// TIA Portal project "SyncProcessi" (V16)

(* hardware
DEVICE "S7-1200 station_1"  S7-1200 Station
   slot 0: "Telaio di montaggio_0"  S7-1200 Rack  Rack  V1.0
   slot 1: "PLC_1"  CPU 1214C DC/DC/DC  6ES7 214-1AG40-0XB0  V4.1
*)

// ===== PLC "PLC_1"  CPU 1214C DC/DC/DC =====

VAR_GLOBAL   // PLC tag table "Tabella delle variabili standard"
   "START_1" AT %I0.0 : Bool;
   "START_2" AT %I0.1 : Bool;
   "STOP_1" AT %I0.2 : Bool;
   "RESTART_2" AT %I0.5 : Bool;
   "OUT_1" AT %Q0.0 : Bool;
   "OUT_2" AT %Q0.1 : Bool;
   "STOP_2" AT %I0.3 : Bool;
   "RESTART_1" AT %I0.4 : Bool;
END_VAR

DATA_BLOCK "VariabiliDiStato_P1"   // DB1
{ S7_Optimized_Access := 'TRUE' }
VERSION : 0.1
   VAR RETAIN
      HOME_1 : Bool := true;
      MOVE : Bool;
      WAIT_1 : Bool;
   END_VAR
BEGIN
END_DATA_BLOCK

DATA_BLOCK "VariabiliDiStato_P2"   // DB2
{ S7_Optimized_Access := 'TRUE' }
VERSION : 0.1
   VAR RETAIN
      HOME_2 : Bool := true;
      ROTATE : Bool;
      WAIT_2 : Bool;
   END_VAR
BEGIN
END_DATA_BLOCK

ORGANIZATION_BLOCK "Main_P1"   // OB1, LAD, ProgramCycle
TITLE = "Main Program Sweep (Cycle)"
{ S7_Optimized_Access := 'TRUE' }
VERSION : 0.1
   VAR_INPUT
      Initial_Call : Bool;   // Initial call of this OB
      Remanence : Bool;   // =True, if remanent data are available
   END_VAR
BEGIN

REGION Network 1
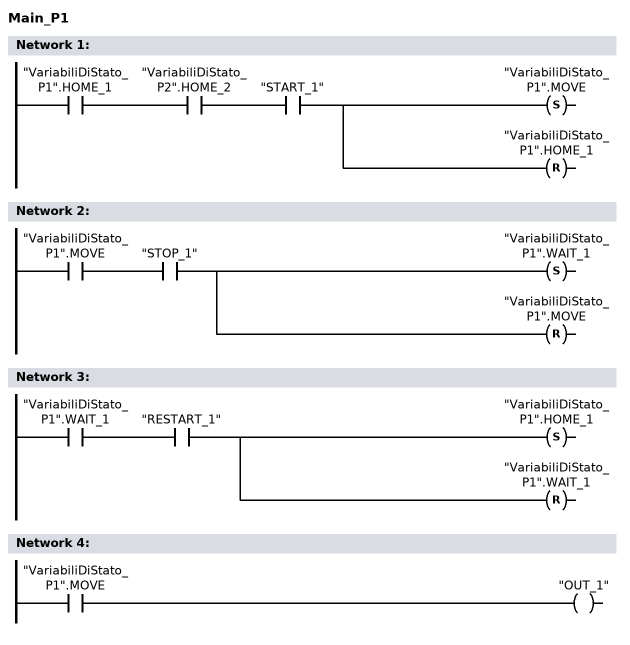
   RUNG wire#powerrail
      Contact( "VariabiliDiStato_P1".HOME_1 )
      Contact( "VariabiliDiStato_P2".HOME_2 )
      Contact( "START_1" )
      wire#w1
      S_Coil( "VariabiliDiStato_P1".MOVE )
   END_RUNG
   RUNG wire#w1
      R_Coil( "VariabiliDiStato_P1".HOME_1 )
   END_RUNG
   // the same network as SCL:
   IF "VariabiliDiStato_P1".HOME_1 AND "VariabiliDiStato_P2".HOME_2 AND "START_1" THEN
       "VariabiliDiStato_P1".MOVE := TRUE;
       "VariabiliDiStato_P1".HOME_1 := FALSE;
   END_IF;
END_REGION

REGION Network 2
   RUNG wire#powerrail
      Contact( "VariabiliDiStato_P1".MOVE )
      Contact( "STOP_1" )
      wire#w1
      S_Coil( "VariabiliDiStato_P1".WAIT_1 )
   END_RUNG
   RUNG wire#w1
      R_Coil( "VariabiliDiStato_P1".MOVE )
   END_RUNG
   // the same network as SCL:
   IF "VariabiliDiStato_P1".MOVE AND "STOP_1" THEN
       "VariabiliDiStato_P1".WAIT_1 := TRUE;
       "VariabiliDiStato_P1".MOVE := FALSE;
   END_IF;
END_REGION

REGION Network 3
   RUNG wire#powerrail
      Contact( "VariabiliDiStato_P1".WAIT_1 )
      Contact( "RESTART_1" )
      wire#w1
      S_Coil( "VariabiliDiStato_P1".HOME_1 )
   END_RUNG
   RUNG wire#w1
      R_Coil( "VariabiliDiStato_P1".WAIT_1 )
   END_RUNG
   // the same network as SCL:
   IF "VariabiliDiStato_P1".WAIT_1 AND "RESTART_1" THEN
       "VariabiliDiStato_P1".HOME_1 := TRUE;
       "VariabiliDiStato_P1".WAIT_1 := FALSE;
   END_IF;
END_REGION

REGION Network 4
   RUNG wire#powerrail
      Contact( "VariabiliDiStato_P1".MOVE )
      Coil( "OUT_1" )
   END_RUNG
   // the same network as SCL:
   "OUT_1" := "VariabiliDiStato_P1".MOVE;
END_REGION
END_ORGANIZATION_BLOCK

ORGANIZATION_BLOCK "Main_P2"   // OB123, LAD, ProgramCycle
TITLE = "Main Program Sweep (Cycle)"
{ S7_Optimized_Access := 'TRUE' }
VERSION : 0.1
   VAR_INPUT
      Initial_Call : Bool;   // Initial call of this OB
      Remanence : Bool;   // =True, if remanent data are available
   END_VAR
BEGIN

REGION Network 1
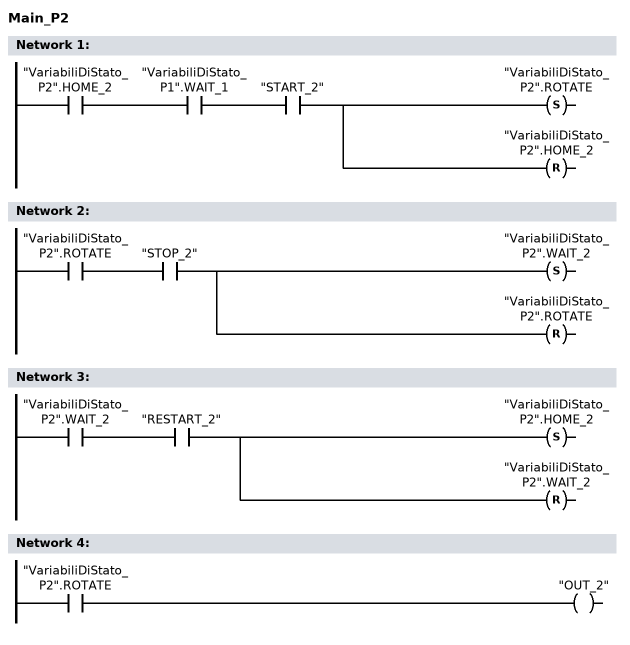
   RUNG wire#powerrail
      Contact( "VariabiliDiStato_P2".HOME_2 )
      Contact( "VariabiliDiStato_P1".WAIT_1 )
      Contact( "START_2" )
      wire#w1
      S_Coil( "VariabiliDiStato_P2".ROTATE )
   END_RUNG
   RUNG wire#w1
      R_Coil( "VariabiliDiStato_P2".HOME_2 )
   END_RUNG
   // the same network as SCL:
   IF "VariabiliDiStato_P2".HOME_2 AND "VariabiliDiStato_P1".WAIT_1 AND "START_2" THEN
       "VariabiliDiStato_P2".ROTATE := TRUE;
       "VariabiliDiStato_P2".HOME_2 := FALSE;
   END_IF;
END_REGION

REGION Network 2
   RUNG wire#powerrail
      Contact( "VariabiliDiStato_P2".ROTATE )
      Contact( "STOP_2" )
      wire#w1
      S_Coil( "VariabiliDiStato_P2".WAIT_2 )
   END_RUNG
   RUNG wire#w1
      R_Coil( "VariabiliDiStato_P2".ROTATE )
   END_RUNG
   // the same network as SCL:
   IF "VariabiliDiStato_P2".ROTATE AND "STOP_2" THEN
       "VariabiliDiStato_P2".WAIT_2 := TRUE;
       "VariabiliDiStato_P2".ROTATE := FALSE;
   END_IF;
END_REGION

REGION Network 3
   RUNG wire#powerrail
      Contact( "VariabiliDiStato_P2".WAIT_2 )
      Contact( "RESTART_2" )
      wire#w1
      S_Coil( "VariabiliDiStato_P2".HOME_2 )
   END_RUNG
   RUNG wire#w1
      R_Coil( "VariabiliDiStato_P2".WAIT_2 )
   END_RUNG
   // the same network as SCL:
   IF "VariabiliDiStato_P2".WAIT_2 AND "RESTART_2" THEN
       "VariabiliDiStato_P2".HOME_2 := TRUE;
       "VariabiliDiStato_P2".WAIT_2 := FALSE;
   END_IF;
END_REGION

REGION Network 4
   RUNG wire#powerrail
      Contact( "VariabiliDiStato_P2".ROTATE )
      Coil( "OUT_2" )
   END_RUNG
   // the same network as SCL:
   "OUT_2" := "VariabiliDiStato_P2".ROTATE;
END_REGION
END_ORGANIZATION_BLOCK